# EPICS autosave request: iocBoot/iocARAmp/auto_settings_ARAmp75A400.req
file "aramp_settings_75A400.req",                P=$(P),  R=$(R)
